(* IEC 61131-3 sources: CodesysTest/alpha/export/PackML/OMAC/Interfaces/IUnitMode.itf/Commands, 10 files *)

(* ---- Abort.m.st ---- *)
(*#-#-#-#-#-#-#-#-#-#---Declaration---#-#-#-#-#-#-#-#-#-#-#-#-#*)

METHOD Abort : BOOL
VAR_INPUT
END_VAR

(* ---- ActingStateCompleted.m.st ---- *)
(*#-#-#-#-#-#-#-#-#-#---Declaration---#-#-#-#-#-#-#-#-#-#-#-#-#*)

METHOD ActingStateCompleted : BOOL
VAR_INPUT
END_VAR

(* ---- Clear.m.st ---- *)
(*#-#-#-#-#-#-#-#-#-#---Declaration---#-#-#-#-#-#-#-#-#-#-#-#-#*)

METHOD Clear : BOOL
VAR_INPUT
END_VAR

(* ---- Hold.m.st ---- *)
(*#-#-#-#-#-#-#-#-#-#---Declaration---#-#-#-#-#-#-#-#-#-#-#-#-#*)

METHOD Hold : BOOL
VAR_INPUT
END_VAR

(* ---- Reset.m.st ---- *)
(*#-#-#-#-#-#-#-#-#-#---Declaration---#-#-#-#-#-#-#-#-#-#-#-#-#*)

METHOD Reset : BOOL
VAR_INPUT
END_VAR

(* ---- Start.m.st ---- *)
(*#-#-#-#-#-#-#-#-#-#---Declaration---#-#-#-#-#-#-#-#-#-#-#-#-#*)

METHOD Start : BOOL
VAR_INPUT
END_VAR

(* ---- Stop.m.st ---- *)
(*#-#-#-#-#-#-#-#-#-#---Declaration---#-#-#-#-#-#-#-#-#-#-#-#-#*)

METHOD Stop : BOOL
VAR_INPUT
END_VAR

(* ---- Suspend.m.st ---- *)
(*#-#-#-#-#-#-#-#-#-#---Declaration---#-#-#-#-#-#-#-#-#-#-#-#-#*)

METHOD Suspend : BOOL
VAR_INPUT
END_VAR

(* ---- Unhold.m.st ---- *)
(*#-#-#-#-#-#-#-#-#-#---Declaration---#-#-#-#-#-#-#-#-#-#-#-#-#*)

METHOD Unhold : BOOL
VAR_INPUT
END_VAR

(* ---- UnSuspend.m.st ---- *)
(*#-#-#-#-#-#-#-#-#-#---Declaration---#-#-#-#-#-#-#-#-#-#-#-#-#*)

METHOD UnSuspend : BOOL
VAR_INPUT
END_VAR
